FUNCTION_BLOCK FB_MoverSectorInterface
VAR
	stSectorConfig			: ST_TrackSectorConfig;	
	refXtsMover				: Tc3_XTS_Utility.ST_PositionInfo;
	refPlanarMover			: MoverSort;
	stTrackSectorStatus		: ST_TrackSectorStatus;
END_VAR

stTrackSectorStatus.MoverIsOnSector	:= _M_IsOnSector();

METHOD PROTECTED _M_IsOnSector : BOOL
_M_IsOnSector	:= (refXtsMover.nTrackObjectid = stSectorConfig.XtsTrackObjId) AND
					IsBetween(value := refXtsMover.fTrackPosition, 
								minV := stSectorConfig.SectorStartPosn, 
								maxV := stSectorConfig.SectorEndPosn);
END_METHOD

PROPERTY P_PlanarMover : REFERENCE TO MoverSort
GET
P_PlanarMover	REF= refPlanarMover;
END_GET
END_PROPERTY

PROPERTY P_SectorStatus : REFERENCE TO ST_TrackSectorStatus
GET
P_SectorStatus	REF= stTrackSectorStatus;
END_GET
END_PROPERTY

PROPERTY P_TrackSectorConfig : REFERENCE TO ST_TrackSectorConfig
GET
P_TrackSectorConfig REF= stSectorConfig;
END_GET
END_PROPERTY

PROPERTY P_XtsPositionInfo : REFERENCE TO Tc3_XTS_Utility.ST_PositionInfo
GET
P_XtsPositionInfo REF= refXtsMover;
END_GET
END_PROPERTY

END_FUNCTION_BLOCK

(* stored: Version 1.1.0.1
   POU FB_MoverSectorInterface: Id {454c8ee6-eb93-03bb-3d09-d82885cc2db0}, SpecialFunc None
   Method _M_IsOnSector: Id {6fb38ca4-6b76-0afd-297f-a5f43cfa3834}
   Property P_PlanarMover: Id {c0ac9430-b382-04fd-3b6a-1962bd5a1c7e}
   Get Get: Id {804e0c8f-06ff-09a3-09d5-b11c0f048c58}
   Property P_SectorStatus: Id {5f8e870d-e32a-0163-2da9-1a6a40e1a497}
   Get Get: Id {de3ffc99-936a-0b5d-0ea1-4e9664bc445a}
   Property P_TrackSectorConfig: Id {5b7ff01c-1c59-02c5-1dcb-4c860620dc5f}
   Get Get: Id {6f251efa-6799-0ba7-38f2-aa9f1e2ed41e}
   Property P_XtsPositionInfo: Id {d96f07f7-f866-0c16-0900-c47c81882126}
   Get Get: Id {ae45bb6f-f61b-08ea-11d8-d62f8182115f} *)
